{attribute 'qualified_only'}
{attribute 'strict'}
TYPE EFeedbackMsgPhotoLumChuck :
(
	WaferPresenceMsg := 10,
	IsInLoadingPositionMsg
);
END_TYPE

(* stored: Version 1.1.0.1, ProductVersion 3.1.4024.12
   DUT EFeedbackMsgPhotoLumChuck: Id {b006c7c0-fc9b-4021-bed6-f993df0abb97} *)
